FUNCTION_BLOCK FB_InterlockHandler
VAR_INPUT
	i_stInterlockList : ST_InterlockList;
END_VAR
VAR
	s_bInterlocked : BOOL;
	s_sReason : STRING(GVL.g_MAX_LEN_INTERLOCK_REASON);
	i : USINT;
	s_nInterlockCnt : USINT;
	
	s_ton : TON;
	s_nIndexShow : USINT := 0;
END_VAR


s_bInterlocked := FALSE;
s_sReason := '';
s_nInterlockCnt := 0;

//Old code showing only one (first found reson)
FOR i := 0 TO (GVL.g_LEN_INTERLOCK_LIST-1) DO
	IF i_stInterlockList.arr_Interlocks[i].bState THEN
		s_bInterlocked := i_stInterlockList.arr_Interlocks[i].bState;
		s_sReason := i_stInterlockList.arr_Interlocks[i].sReason;
		EXIT;
	END_IF
END_FOR

//**FOR i := 0 TO (GVL.g_LEN_INTERLOCK_LIST-1) DO
//**	IF i_stInterlockList.arr_Interlocks[i].bState THEN
//**		s_nInterlockCnt := s_nInterlockCnt + 1;
//**		s_bInterlocked := i_stInterlockList.arr_Interlocks[i].bState;
//**		IF s_nInterlockCnt > 1 THEN
//**			s_sReason := CONCAT(s_sReason, CONCAT('; ', i_stInterlockList.arr_Interlocks[i].sReason));
//**		ELSE
//**			s_sReason := i_stInterlockList.arr_Interlocks[i].sReason;
//**		END_IF	
//**	END_IF
//**END_FOR

//New code showing all active interlocks time based
(*
	s_ton(IN := NOT(s_ton.Q), PT := T#2S);

	IF s_ton.Q THEN
		IF i_stInterlockList.arr_Interlocks[s_nIndexShow].bState THEN
			s_bInterlocked := i_stInterlockList.arr_Interlocks[s_nIndexShow].bState;
			s_sReason := i_stInterlockList.arr_Interlocks[s_nIndexShow].sReason;
		END_IF
		
		IF s_nIndexShow < (GVL.g_LEN_INTERLOCK_LIST-1) THEN
			s_nIndexShow := s_nIndexShow + 1; 
		ELSE
			s_nIndexShow := 0;
		END_IF
		
	END_IF
*)

PROPERTY PUBLIC p_bInterlocked : BOOL
GET

p_bInterlocked := s_bInterlocked;
END_GET
END_PROPERTY

PROPERTY PUBLIC p_sReason : STRING
GET

p_sReason := s_sReason;
END_GET
END_PROPERTY

END_FUNCTION_BLOCK

(* stored: Version 1.1.0.1, ProductVersion 3.1.4024.12
   POU FB_InterlockHandler: Id {3f803ac0-c811-44d7-bc37-de6385932f87}, SpecialFunc None
   Property p_bInterlocked: Id {86e04223-6d35-4c0b-a8e3-7fa2c5ae859f}
   Get Get: Id {18a6c684-2c70-43a4-813f-00bd04500324}
   Property p_sReason: Id {aaf90641-7dc3-4684-ad11-173ff784777c}
   Get Get: Id {dcfe3acf-6a85-4f02-8995-d2803f5f511d} *)
